FUNCTION_BLOCK TcoAnalogueInspectorTests EXTENDS TcoInspectorTests
VAR
    _sut            : TcoInspectors.TcoAnalogueInspector(THIS^);
    _inspectedValue : LREAL;
END_VAR

METHOD Inspect : TcoInspectors.IInspector
Inspect := _sut.Inspect(_inspectedValue);
END_METHOD

METHOD PROTECTED Main
SUPER^.Main();
END_METHOD

METHOD  WithCoordinator : REFERENCE TO TcoInspectorTests
VAR_INPUT
	inoCoordinator : TcoCore.ITcoCoordinator;
END_VAR
_sut.WithCoordinator(_coordinator);
WithCoordinator REF= THIS^;
END_METHOD

END_FUNCTION_BLOCK

(* stored: Version 1.1.0.1, ProductVersion 3.1.4024.9
   POU TcoAnalogueInspectorTests: Id {8dc99e3a-e964-0734-3e39-363ce73c5757}, SpecialFunc None
   Method Inspect: Id {3703065d-567a-0583-2b5d-991c71f6123a}
   Method Main: Id {060cfbf3-cf54-0d00-1452-4a68e42aa954}
   Method WithCoordinator: Id {9d0edf65-b764-0fe1-0ea6-c44ac1de6e92} *)
